FUNCTION_BLOCK EcMasterProtocolError IMPLEMENTS IEcTask
VAR_INPUT
END_VAR
VAR_OUTPUT
END_VAR
VAR
	iState : INT;
	masterProtocolErr : Tc2_EtherCAT.FB_EcGetLastProtErrInfo;
	_execute: BOOL;
	_done: BOOL;
	_busy: BOOL;
	_error: BOOL;
	_netId: AMSNETID;
END_VAR

CASE iState OF
	0:
		IF _execute THEN
			_done := FALSE;
			_busy := TRUE;
			_error := FALSE;
			masterProtocolErr.bExecute := TRUE;
			IF masterProtocolErr.bBusy THEN
				iState := 10;
				_execute := false;
			END_IF
		END_IF
	10:
		IF NOT masterProtocolErr.bBusy THEN
			IF NOT masterProtocolErr.bError THEN
				_done := TRUE;
			ELSE
				_error := TRUE;
			END_IF
			_busy := FALSE;
			masterProtocolErr.bExecute := FALSE;
			iState := 0;
		END_IF
END_CASE

masterProtocolErr(sNetId := Tc2_System.F_CreateAmsNetId(nIds := NetId));

{warning 'add method implementation '}
METHOD Abort : BOOL
masterProtocolErr.bExecute := FALSE;
_busy := FALSE;
_execute := FALSE;
Abort := TRUE;
iState := 0;
END_METHOD

{warning 'add property implementation'}
PROPERTY Busy : BOOL
GET
Busy := _busy;
END_GET
END_PROPERTY

PROPERTY DeviceAddr : uint
GET
DeviceAddr := masterProtocolErr.nSlaveAddr;
END_GET
SET
masterProtocolErr.nSlaveAddr := DeviceAddr;
END_SET
END_PROPERTY

{warning 'add property implementation'}
PROPERTY Done : BOOL
GET
Done := _done;
END_GET
END_PROPERTY

{warning 'add property implementation'}
PROPERTY Error : BOOL
GET
Error := _error;
END_GET
END_PROPERTY

{warning 'add method implementation '}
METHOD Execute : BOOL
IF NOT masterProtocolErr.bBusy THEN
	Execute := _execute := TRUE;
END_IF
END_METHOD

PROPERTY LastProtocolError : ST_EcLastProtErrInfo
GET
LastProtocolError := masterProtocolErr.info;
END_GET
END_PROPERTY

{warning 'add property implementation'}
PROPERTY NetID : amsnetid
GET
NetID := _netId;
END_GET
SET
_netId := NetID;
END_SET
END_PROPERTY

PROPERTY ProtocolType : E_EcMbxProtType
GET
ProtocolType := masterProtocolErr.eProtocol;
END_GET
SET
masterProtocolErr.eProtocol := ProtocolType;
END_SET
END_PROPERTY

END_FUNCTION_BLOCK

(* stored: Version 1.1.0.1, ProductVersion 3.1.4024.9
   POU EcMasterProtocolError: Id {524c00f0-8a88-44a2-a6fb-3d2ba1f9f6ba}, SpecialFunc None
   Method Abort: Id {8ec4446a-8d45-4969-9dd2-5ba4f2d9caab}
   Property Busy: Id {e5cefaca-c9a0-41a0-b3e8-81ea42f3144e}
   Get Get: Id {dcf3342c-b43b-4ead-87bb-ae8ac7bcdd07}
   Property DeviceAddr: Id {1fe96107-23d1-4b5f-88a7-ad0b59942e77}
   Get Get: Id {436c9308-645c-4c39-94f1-40e27366e4b9}
   Set Set: Id {81e3897f-c809-42cf-8734-22737817bc77}
   Property Done: Id {af1c7502-3456-43b4-a8b2-d7e4a828e042}
   Get Get: Id {84f7f587-6f91-4f2a-8381-f97151a79748}
   Property Error: Id {f4aa0eb9-79e4-409b-b2e1-ac12ecdb9de9}
   Get Get: Id {bd234570-99a0-4475-a923-7b015eea83ff}
   Method Execute: Id {62fd5f42-f783-4971-b219-17e2c65efc93}
   Property LastProtocolError: Id {97994ea7-26e7-4268-a85a-b58c1a4b746f}
   Get Get: Id {b632c0cb-a710-4c42-8add-3986abf7a4aa}
   Property NetID: Id {5deb011a-19dd-404b-be13-e964c030b2a7}
   Get Get: Id {b400f4fb-8496-4e0f-ac88-82b48cd45add}
   Set Set: Id {5ea57270-e776-43cb-b3ca-37dd1ea79d51}
   Property ProtocolType: Id {43f17fdc-415f-48ab-9339-c61e728b4827}
   Get Get: Id {fc7eb7bc-1cab-410a-ae7d-f7e843f8900b}
   Set Set: Id {fbfd0e40-586a-4862-8a6f-ec86006ff0d2} *)
